// TIA Portal V20 export
VAR_GLOBAL   // PLC tag table "LibraryObjects"
END_VAR
VAR_GLOBAL CONSTANT   // user constants
   LAF_DRV_DIAG_SINA_TYPE_S120_EPOS : UInt := 125;   // Type of SINAMICS is S120 with EPOS
   LAF_DRV_DIAG_SINA_TYPE_NO_TYPE : UInt := 0;   // Type of SINAMICS is not specified
   LAF_DRV_DIAG_SINA_TYPE_G120 : UInt := 114;   // Type of SINAMICS is G120
   LAF_DRV_DIAG_SINA_TYPE_S210_EPOS : UInt := 223;   // Type of SINAMICS is S210 with EPOS
   LAF_DRV_DIAG_NO_DO : UDInt := 41;   // Number of drive objects for drive diagnostic
   LAF_DRV_DIAG_SINA_TYPE_S210 : UInt := 222;   // Type of SINAMICS is S210
   LAF_DRV_DIAG_SINA_TYPE_S120 : UInt := 124;   // Type of SINAMICS is S120
   LAF_DRV_DIAG_SINA_TYPE_S200 : UInt := 220;   // Type of SINAMICS is S200
   LAF_DRV_DIAG_SINA_TYPE_S200_EPOS : UInt := 221;   // Type of SINAMICS is S200 with EPOS
   LAF_DRV_DIAG_AXIS_NO_AXIS : DB_ANY := 0;   // No Technology Object used
END_VAR
